PROGRAM MAIN
VAR
	fbDev1	:	FB_ExampleDevice;
	
	BP1	:	ST_BeamParams;
	BP2	:	ST_BeamParams;
	Test	:	BOOL;
	
	rtInit	:	R_TRIG;
	Initialize	:	BOOL := TRUE;
	
END_VAR

//Sub-system Device PLC
// This PLC runs 4 

Test := F_SafeBPCompare(BP1,BP2);

IF Initialize THEN
	fbDev1.Initialize();
	Initialize := FALSE;
END_IF

//Example devices
fbDev1();

PMPS_Arbiter();

ACTION Initialize:

END_ACTION

END_PROGRAM

(* stored: Version 1.1.0.1, ProductVersion 3.1.4022.12
   POU MAIN: Id {8a7bcfd2-1a2b-4363-aa47-c19391bf1f9c}, SpecialFunc None
   Action Initialize: Id {b0ee480a-3d4b-001d-04c4-43cdc47895c8} *)
